{attribute addProperty BoxType "EL3783-0000-0018"}
{attribute addProperty Id "I1_SamplesAT %I*ARRAY [0..19] OF INT32040"}
{attribute addProperty CRC "1102457989"}
{attribute addProperty SizeInBites "320"}
{attribute addProperty SizeInBytes "40"}
TYPE L1_Current_Samples_41B62C85 :
STRUCT
	{attribute addProperty Name "I1_Samples"}
	I1_Samples AT %I* : ARRAY [0..19] OF INT;
END_STRUCT
END_TYPE

(* stored: Version 1.2.0.0, ProductVersion 3.1.4024.9
   DUT L1_Current_Samples_41B62C85: Id {5bc8b1b9-bf30-4515-8600-fef783bf6a2e} *)
